/// this is the container of informations that the unit wants to share with the world outside of the PLC
/// This struct should only be read from by external applications.
TYPE MachineComPublish :
STRUCT
  State : ZApplication.UnitStateMachineState; // state the unit is in
  Request : MachineComRequest; // booleans that indictate which action is currently possible to perform with this unit
  Equipment : MachineComPublishEquipment;  // structs for equipment objects which are used by the bridges
END_STRUCT
END_TYPE

(* stored: Version 1.1.0.1
   DUT MachineComPublish: Id {c351db49-bd7d-4ab1-a8b0-d6a9816a85a3} *)
